VAR_GLOBAL
	In_bol_EmergencyOff AT %I* : BOOL; // Emergency Off Button
END_VAR

(* stored: Version 1.1.0.1, ProductVersion 3.1.0.19
   GVL Io: Id {407668e5-83c7-4fef-b1ff-b6c883942ff7} *)
